{attribute 'enable_dynamic_creation'}
FUNCTION_BLOCK FB_Slot
VAR_INPUT
END_VAR
VAR_OUTPUT
END_VAR
VAR
	pOwner	: POINTER TO FB_Object;
	pChild	: POINTER TO FB_Object;
	nNr		: UINT;
	stRelPos: ST_3DPoint;
END_VAR

METHOD FB_init : BOOL
VAR_INPUT
	bInitRetains : BOOL; // if TRUE, the retain variables are initialized (warm start / cold start)
	bInCopyCode : BOOL;  // if TRUE, the instance afterwards gets moved into the copy code (online change)
	pOwner		: POINTER TO FB_Object;
END_VAR
THIS^.pOwner := pOwner;
END_METHOD

PROPERTY P_nNr : UINT
GET
P_nNr := nNr;
END_GET
SET
nNr := P_nNr;
END_SET
END_PROPERTY

PROPERTY P_rRelPosY : REAL
SET
stRelPos.Y := P_rRelPosY;
END_SET
GET
P_rRelPosY := stRelPos.Y;
END_GET
END_PROPERTY

PROPERTY P_rRelPosX : REAL
SET
stRelPos.X := P_rRelPosX;
END_SET
GET
P_rRelPosX := stRelPos.X;
END_GET
END_PROPERTY

PROPERTY P_pChild : POINTER TO FB_Object
GET
P_pChild := pChild;
END_GET
SET
pChild := P_pChild;
END_SET
END_PROPERTY

PROPERTY P_stRelPos : ST_3DPoint
SET
stRelPos := P_stRelPos;
END_SET
GET
P_stRelPos := stRelPos;
END_GET
END_PROPERTY

PROPERTY P_stAbsPos : ST_3DPoint
GET
VAR
	stTemp : ST_3DPoint;
	pMzTool: POINTER TO FB_MzTool;
	pTarget: POINTER TO FB_TargetBase;
END_VAR
IF pOwner^.P_eObjectType = E_ObjectType.OBJECTTYPE_MZHead THEN
	pMzTool := pOwner;
	stTemp := pMzTool^.P_stAbsPosTotal;
	stTemp.X := stTemp.X + stRelPos.X;
	stTemp.Y := stTemp.Y + stRelPos.Y;
	P_stAbsPos := stTemp;
ELSIF pOwner^.M_bIsGroup(E_ObjectGroup.OBJECTGROUP_MzTool) THEN
	pMzTool := pOwner;
	P_stAbsPos := F_Add3DPoints(stRelPos, pMzTool^.P_stAbsPosPhysExclPiece);
ELSIF pOwner^.M_bIsGroup(E_ObjectGroup.OBJECTGROUP_Target) THEN
	pTarget := pOwner;
	P_stAbsPos := F_Add3DPoints(stRelPos, pTarget^.P_stAbsPosLB);
END_IF
END_GET
END_PROPERTY

PROPERTY P_rRelPosZ : REAL
GET
P_rRelPosZ := stRelPos.Z;
END_GET
SET
stRelPos.Z := P_rRelPosZ;
END_SET
END_PROPERTY

END_FUNCTION_BLOCK

(* stored: Version 1.1.0.1, ProductVersion 3.1.4020.12
   POU FB_Slot: Id {e24cb34c-9386-4766-bfb6-60ee8362a2de}, SpecialFunc None
   Method FB_init: Id {21833cee-547c-4a11-aa16-b4eb0d1e6b45}
   Property P_nNr: Id {3c4bd464-9797-42b2-8074-0b1f4a6bf0c1}
   Get Get: Id {5adfd437-6017-4f7c-a710-e0c96a476711}
   Set Set: Id {ce30d8d9-5fb5-4a5f-82bf-9d1ad5166f88}
   Property P_rRelPosY: Id {4fac106b-7284-471c-a554-cd2189e97c22}
   Set Set: Id {a8a33bc6-db5f-4610-8ca0-9f7d9c329ae4}
   Get Get: Id {ac969bc0-fd7e-47db-8206-969126257610}
   Property P_rRelPosX: Id {8cddccde-f83e-4541-a409-9cb93abf12e2}
   Set Set: Id {6dbeea8b-4fd4-49d1-a79c-6d298e9967ac}
   Get Get: Id {a7a910bc-f35d-430d-a1f2-c71783120de4}
   Property P_pChild: Id {93479887-06f8-4ab7-b41f-f57687cb48d7}
   Get Get: Id {67275c62-6da1-43ed-a7ea-4d4128620b4d}
   Set Set: Id {dcf65487-7f25-45ce-b851-b37dc11d831d}
   Property P_stRelPos: Id {d4d3907d-3b0e-47d3-bc09-1ecaffc4d877}
   Set Set: Id {1eea22a1-ea64-4c59-8c9c-1e1d731f6588}
   Get Get: Id {6c631d4a-31eb-4aa7-a318-fe904d96035c}
   Property P_stAbsPos: Id {e157931f-30ac-4d87-b06c-fc63af0ada22}
   Get Get: Id {cf361eac-e23e-4bb8-8d72-954df8946a24}
   Property P_rRelPosZ: Id {ece4cbd0-3458-4d91-b82a-13eb847fdbe9}
   Get Get: Id {86eb722c-0f42-47b6-a9af-0e403a30b481}
   Set Set: Id {b7d736de-7559-49cd-8bbb-3848b5f6bd0f} *)
